FUNCTION_BLOCK FB_Puls
VAR_INPUT
	bReset				: 	BOOL;
	tFlashOn				: 	TIME;
	tFlashOff				: 	TIME;
END_VAR
VAR_OUTPUT
	bFlashEnable			: 	BOOL;
END_VAR
VAR
	tonFlashOn			: 	TON;
	tonFlashOff			: 	TON;
END_VAR

tonFlashOn(IN:= bFlashEnable, PT:= tFlashOn);

tonFlashOff(IN:= NOT bFlashEnable, PT:= tFlashOff);

IF bReset  OR tFlashOn = t#0ms OR tFlashOff = t#0m THEN
	bFlashEnable := FALSE;
ELSE

	IF	tonFlashOn.Q	THEN
		bFlashEnable	:= FALSE;
	END_IF
	
	IF	tonFlashOff.Q	THEN
		bFlashEnable	:= TRUE;
	END_IF
END_IF

END_FUNCTION_BLOCK

(* stored: Version 1.1.0.1, ProductVersion 3.1.4024.15
   POU FB_Puls: Id {feaef9b9-433f-434b-907a-e26615e0589e}, SpecialFunc None *)
